// TIA Portal V17 export
// export: Created 2025-03-05T08:00:07.0490995Z, ExportSetting WithDefaults, DisplayName Totally Integrated Automation Portal, DisplayVersion V17 Update 8, DisplayName TIA Portal Openness, DisplayVersion V17 Update 8, DisplayName TIA Portal Version Control Interface, DisplayVersion V17, DisplayName SINAMICS Startdrive Advanced, DisplayVersion V17 SP2, DisplayName SINAMICS Startdrive G110M, G120, G120C, G120D, G120P, G115D, DisplayVersion V17 SP2, DisplayName SINAMICS Startdrive G130, G150, S120, S150, SINAMICS MV, S210, DisplayVersion V17 SP2, DisplayName STEP 7 Professional, DisplayVersion V17 Update 8, DisplayName SINUMERIK ONE STEP 7 Toolbox, DisplayVersion V17 Update 12, DisplayName SINUMERIK 840D sl STEP 7 Toolbox, DisplayVersion V17 Update 12, DisplayName STEP 7 Safety, DisplayVersion V17 Update 6, DisplayName WinCC Advanced, DisplayVersion V17 Update 8
FUNCTION_BLOCK "FB2002_BA_MODE"   // FB2002, LAD
{ S7_Optimized_Access := 'FALSE' }
VERSION : 0.1
// stored: AutoNumber false, IsIECCheckEnabled false, SetENOAutomatically false, UDAEnableTagReadback false
   VAR_INPUT
      OPTIONS_0 { ExternalAccessible := 'False'; ExternalVisible := 'False'; ExternalWritable := 'False'} : Byte := 2#0000_0000;   // OPTIONS BYTE 0
      BA1_BUTTON_I { ExternalAccessible := 'False'; ExternalVisible := 'False'; ExternalWritable := 'False'} : Bool;   // BA1 BUTTON INPUT
      BA2_BUTTON_I { ExternalAccessible := 'False'; ExternalVisible := 'False'; ExternalWritable := 'False'} : Bool;   // BA2 BUTTON INPUT
      BA3_BUTTON_I { ExternalAccessible := 'False'; ExternalVisible := 'False'; ExternalWritable := 'False'} : Bool;   // BA3 BUTTON INPUT
      BA5_BUTTON_I { ExternalAccessible := 'False'; ExternalVisible := 'False'; ExternalWritable := 'False'} : Bool;   // BA5 BUTTON INPUT
      SAFETY_ENABLED_W_DOOR_OPENED { ExternalAccessible := 'False'; ExternalVisible := 'False'; ExternalWritable := 'False'} : Bool;   // SAFETY ENABLED WITH DOOR OPENED (ENABLING DEVICE AND HT10 ENABLE BUTTON)
      SAFETY_GATES_CLSD_AND_LCKD { ExternalAccessible := 'False'; ExternalVisible := 'False'; ExternalWritable := 'False'} : Bool;   // SAFETY GATES CLOSED AND LOCKED
      START_SERVICES_GLOBAL { ExternalAccessible := 'False'; ExternalVisible := 'False'; ExternalWritable := 'False'} : Bool;   // START SERVICES GLOBAL
      ANY_MCH_CYCLE_RUN { ExternalAccessible := 'False'; ExternalVisible := 'False'; ExternalWritable := 'False'} : Bool;   // ANY MACHINE CYCLE RUNNING
      MCH_RESET_FAULTS { ExternalAccessible := 'False'; ExternalVisible := 'False'; ExternalWritable := 'False'} : Bool;   // MACHINE_RESET_FAULTS
   END_VAR
   VAR_OUTPUT
      NO_BA_MODE_SLCTD_WRN { ExternalAccessible := 'False'; ExternalVisible := 'False'; ExternalWritable := 'False'} : Bool;   // NO BA MODE SELECTED WARNING
      CHANGE_TO_BA1_MODE_WRN { ExternalAccessible := 'False'; ExternalVisible := 'False'; ExternalWritable := 'False'} : Bool;   // CHANGE TO BA1 MODE WARNING
      CHANGE_TO_BA2_MODE_WRN { ExternalAccessible := 'False'; ExternalVisible := 'False'; ExternalWritable := 'False'} : Bool;   // CHANGE TO BA2 MODE WARNING
      CHANGE_TO_BA3_MODE_WRN { ExternalAccessible := 'False'; ExternalVisible := 'False'; ExternalWritable := 'False'} : Bool;   // CHANGE TO BA3 MODE WARNING
      CHANGE_TO_BA5_MODE_WRN { ExternalAccessible := 'False'; ExternalVisible := 'False'; ExternalWritable := 'False'} : Bool;   // CHANGE TO BA5 MODE WARNING
      BA1_MODE_LED_O { ExternalAccessible := 'False'; ExternalVisible := 'False'; ExternalWritable := 'False'} : Bool;   // BA1 MODE BUTTON LED OUTPUT
      BA2_MODE_LED_O { ExternalAccessible := 'False'; ExternalVisible := 'False'; ExternalWritable := 'False'} : Bool;   // BA2 MODE BUTTON LED OUTPUT
      BA3_MODE_LED_O { ExternalAccessible := 'False'; ExternalVisible := 'False'; ExternalWritable := 'False'} : Bool;   // BA3 MODE BUTTON LED OUTPUT
   END_VAR
   VAR_IN_OUT
      MODE_GROUP_GENERAL_DB : "AUTO_SINGLE_SEMI_MANUAL";
      MODE_GROUP_BA_DB : "BA_MODE";
   END_VAR
   VAR_TEMP
      INPUTS_MASK : Byte;   // INPUT MASK
      O_BYTE_0 : Struct   // OPTIONS BYTE 0
         BA_BUTTONS : Bool;   // BA MODE BUTTONS OPTION
         CHANGE_MODE_SEOC_ALARM : Bool;   // CHANGE MODE SEOC ALARM OPTION
         MODE_SELECTED_MEMORY : Bool;   // MODE SELECTED MEMORY OPTION
         SPARE : Bool;
         SPARE_1 : Bool;
         SPARE_2 : Bool;
         SPARE_3 : Bool;
         SPARE_4 : Bool;
      END_STRUCT;
      DB_NUMBER : DInt;   // DB NUMBER FOR ALARM DECODING
   END_VAR
   VAR_TEMP   // added for the SCL form of the ladder/FBD networks
      _w1 : Bool;
      _w2 : Bool;
   END_VAR
BEGIN

NETWORK
TITLE = READ INSTANCE DB
      L     DINO;
      +     10#800000;
      T     #DB_NUMBER;


REGION Network 2: OPTIONS
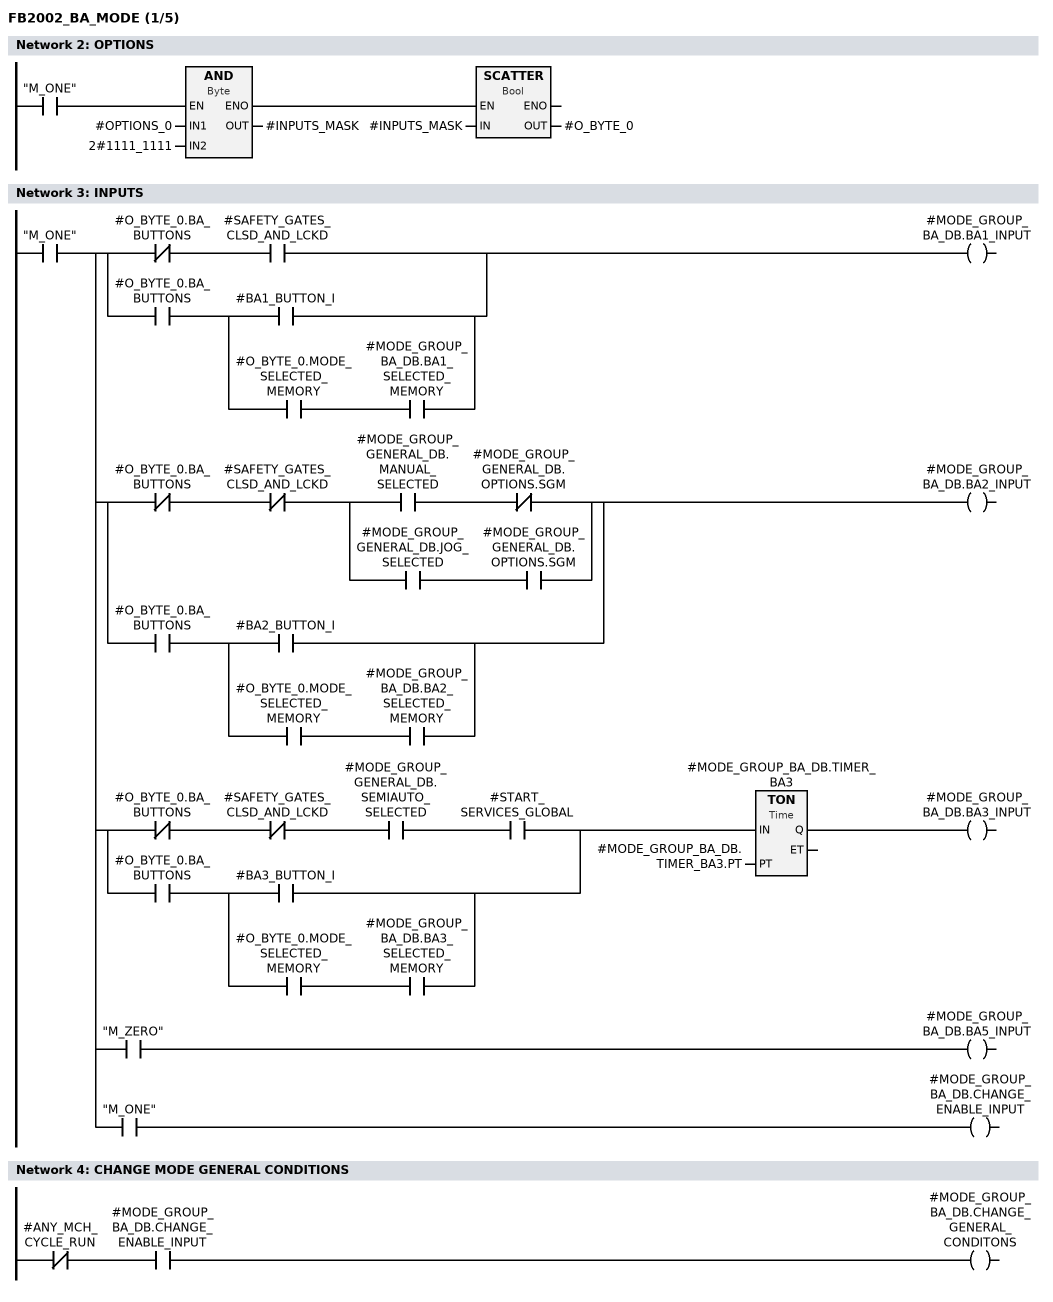
   RUNG wire#powerrail
      Contact( "M_ONE" )
      { S7_Templates := "SrcType := Byte"; S7_GenerateENO := "TRUE" } And(in1 := #OPTIONS_0, in2 := 2#1111_1111, out => #INPUTS_MASK)
      { S7_Templates := "[dest_type := Bool, src_type := Byte]" } SCATTER(IN := #INPUTS_MASK, OUT => #O_BYTE_0)
   END_RUNG
   // the same network as SCL:
   IF "M_ONE" THEN
       #INPUTS_MASK := #OPTIONS_0 AND 2#1111_1111;
       SCATTER(IN := #INPUTS_MASK, OUT => #O_BYTE_0);
   END_IF;
END_REGION

REGION Network 3: INPUTS
   RUNG wire#powerrail
      Contact( "M_ONE" )
      wire#w1
      I_Contact( #O_BYTE_0.BA_BUTTONS )
      Contact( #SAFETY_GATES_CLSD_AND_LCKD )
      wire#w2
      Coil( #MODE_GROUP_BA_DB.BA1_INPUT )
   END_RUNG
   RUNG wire#w1
      Contact( #O_BYTE_0.BA_BUTTONS )
      wire#w3
      Contact( #BA1_BUTTON_I )
   END_RUNG wire#w2
   RUNG wire#w3
      Contact( #O_BYTE_0.MODE_SELECTED_MEMORY )
      Contact( #MODE_GROUP_BA_DB.BA1_SELECTED_MEMORY )
   END_RUNG wire#w2
   RUNG wire#w1
      I_Contact( #O_BYTE_0.BA_BUTTONS )
      I_Contact( #SAFETY_GATES_CLSD_AND_LCKD )
      wire#w4
      Contact( #MODE_GROUP_GENERAL_DB.MANUAL_SELECTED )
      I_Contact( #MODE_GROUP_GENERAL_DB.OPTIONS.SGM )
      wire#w5
      Coil( #MODE_GROUP_BA_DB.BA2_INPUT )
   END_RUNG
   RUNG wire#w4
      Contact( #MODE_GROUP_GENERAL_DB.JOG_SELECTED )
      Contact( #MODE_GROUP_GENERAL_DB.OPTIONS.SGM )
   END_RUNG wire#w5
   RUNG wire#w1
      Contact( #O_BYTE_0.BA_BUTTONS )
      wire#w6
      Contact( #BA2_BUTTON_I )
   END_RUNG wire#w5
   RUNG wire#w6
      Contact( #O_BYTE_0.MODE_SELECTED_MEMORY )
      Contact( #MODE_GROUP_BA_DB.BA2_SELECTED_MEMORY )
   END_RUNG wire#w5
   RUNG wire#w1
      I_Contact( #O_BYTE_0.BA_BUTTONS )
      I_Contact( #SAFETY_GATES_CLSD_AND_LCKD )
      Contact( #MODE_GROUP_GENERAL_DB.SEMIAUTO_SELECTED )
      Contact( #START_SERVICES_GLOBAL )
      wire#w7
      { S7_Templates := "time_type := Time" } #MODE_GROUP_BA_DB.TIMER_BA3.TON(pt := #MODE_GROUP_BA_DB.TIMER_BA3.PT, et =>)
      Coil( #MODE_GROUP_BA_DB.BA3_INPUT )
   END_RUNG
   RUNG wire#w1
      Contact( #O_BYTE_0.BA_BUTTONS )
      wire#w8
      Contact( #BA3_BUTTON_I )
   END_RUNG wire#w7
   RUNG wire#w8
      Contact( #O_BYTE_0.MODE_SELECTED_MEMORY )
      Contact( #MODE_GROUP_BA_DB.BA3_SELECTED_MEMORY )
   END_RUNG wire#w7
   RUNG wire#w1
      Contact( "M_ZERO" )
      Coil( #MODE_GROUP_BA_DB.BA5_INPUT )
   END_RUNG
   RUNG wire#w1
      Contact( "M_ONE" )
      Coil( #MODE_GROUP_BA_DB.CHANGE_ENABLE_INPUT )
   END_RUNG
   // the same network as SCL:
   #MODE_GROUP_BA_DB.BA1_INPUT := "M_ONE" AND ((NOT #O_BYTE_0.BA_BUTTONS AND #SAFETY_GATES_CLSD_AND_LCKD) OR (#O_BYTE_0.BA_BUTTONS AND (#BA1_BUTTON_I OR (#O_BYTE_0.MODE_SELECTED_MEMORY AND #MODE_GROUP_BA_DB.BA1_SELECTED_MEMORY))));
   #MODE_GROUP_BA_DB.BA2_INPUT := "M_ONE" AND ((NOT #O_BYTE_0.BA_BUTTONS AND NOT #SAFETY_GATES_CLSD_AND_LCKD AND ((#MODE_GROUP_GENERAL_DB.MANUAL_SELECTED AND NOT #MODE_GROUP_GENERAL_DB.OPTIONS.SGM) OR (#MODE_GROUP_GENERAL_DB.JOG_SELECTED AND #MODE_GROUP_GENERAL_DB.OPTIONS.SGM))) OR (#O_BYTE_0.BA_BUTTONS AND (#BA2_BUTTON_I OR (#O_BYTE_0.MODE_SELECTED_MEMORY AND #MODE_GROUP_BA_DB.BA2_SELECTED_MEMORY))));
   #MODE_GROUP_BA_DB.TIMER_BA3.TON(IN := "M_ONE" AND ((NOT #O_BYTE_0.BA_BUTTONS AND NOT #SAFETY_GATES_CLSD_AND_LCKD AND #MODE_GROUP_GENERAL_DB.SEMIAUTO_SELECTED AND #START_SERVICES_GLOBAL) OR (#O_BYTE_0.BA_BUTTONS AND (#BA3_BUTTON_I OR (#O_BYTE_0.MODE_SELECTED_MEMORY AND #MODE_GROUP_BA_DB.BA3_SELECTED_MEMORY)))),
                           PT := #MODE_GROUP_BA_DB.TIMER_BA3.PT);
   #MODE_GROUP_BA_DB.BA3_INPUT := #MODE_GROUP_BA_DB.TIMER_BA3.Q;
   #MODE_GROUP_BA_DB.BA5_INPUT := "M_ONE" AND "M_ZERO";
   #MODE_GROUP_BA_DB.CHANGE_ENABLE_INPUT := "M_ONE" AND "M_ONE";
END_REGION

REGION Network 4: CHANGE MODE GENERAL CONDITIONS
   RUNG wire#powerrail
      I_Contact( #ANY_MCH_CYCLE_RUN )
      Contact( #MODE_GROUP_BA_DB.CHANGE_ENABLE_INPUT )
      Coil( #MODE_GROUP_BA_DB.CHANGE_GENERAL_CONDITONS )
   END_RUNG
   // the same network as SCL:
   #MODE_GROUP_BA_DB.CHANGE_GENERAL_CONDITONS := NOT #ANY_MCH_CYCLE_RUN AND #MODE_GROUP_BA_DB.CHANGE_ENABLE_INPUT;
END_REGION

REGION Network 5: OPERATOR HELP
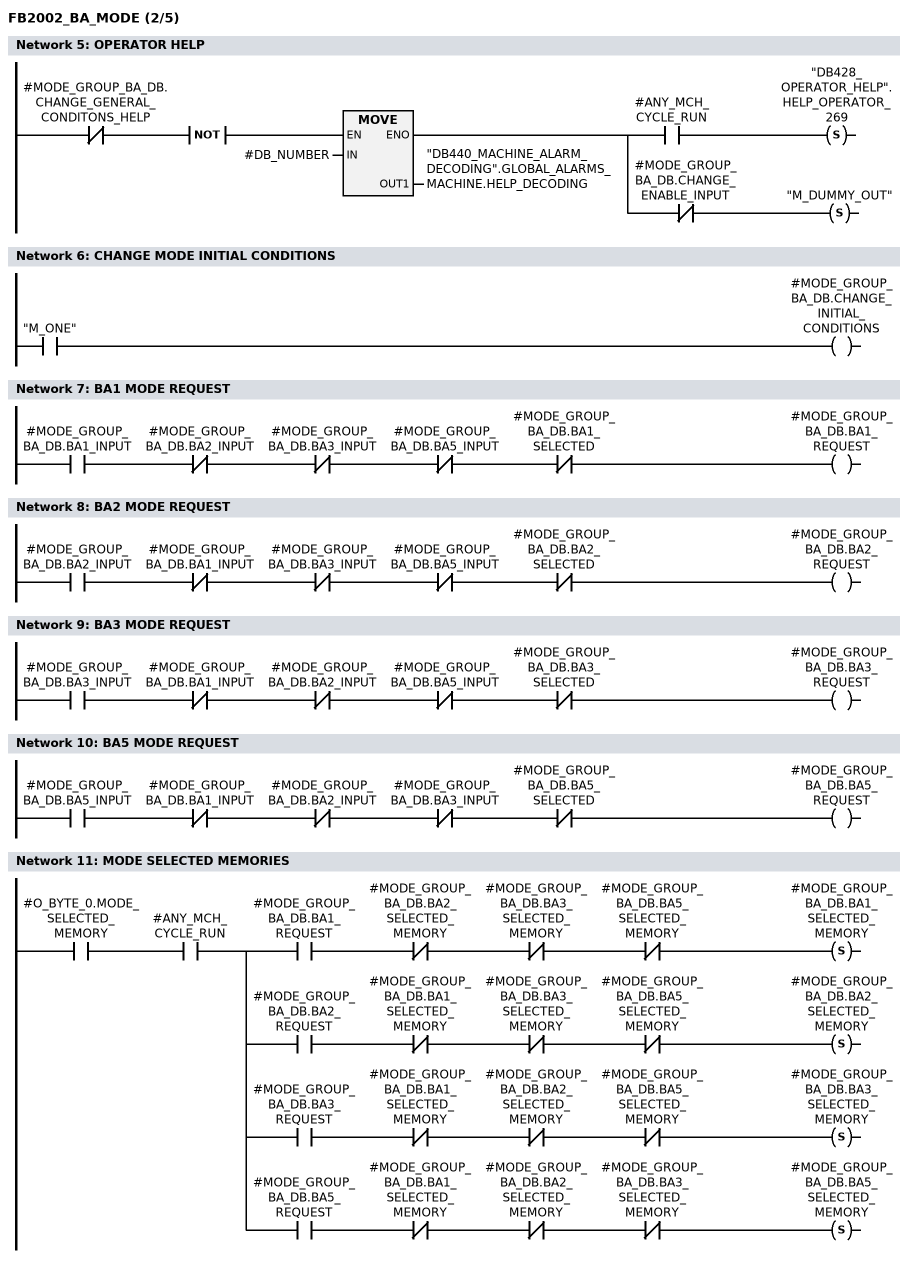
   RUNG wire#powerrail
      I_Contact( #MODE_GROUP_BA_DB.CHANGE_GENERAL_CONDITONS_HELP )
      Not()
      { S7_GenerateENO := "TRUE" } Move(in := #DB_NUMBER, out1 => "DB440_MACHINE_ALARM_DECODING".GLOBAL_ALARMS_MACHINE.HELP_DECODING)
      wire#w1
      Contact( #ANY_MCH_CYCLE_RUN )
      S_Coil( "DB428_OPERATOR_HELP".HELP_OPERATOR_269 )
   END_RUNG
   RUNG wire#w1
      I_Contact( #MODE_GROUP_BA_DB.CHANGE_ENABLE_INPUT )
      S_Coil( "M_DUMMY_OUT" )
   END_RUNG
   // the same network as SCL:
   // ENO of a box is taken as its EN; it also drops when the box reports an error
   #_w1 := NOT (NOT #MODE_GROUP_BA_DB.CHANGE_GENERAL_CONDITONS_HELP);
   IF #_w1 THEN "DB440_MACHINE_ALARM_DECODING".GLOBAL_ALARMS_MACHINE.HELP_DECODING := #DB_NUMBER; END_IF;
   IF #_w1 AND #ANY_MCH_CYCLE_RUN THEN "DB428_OPERATOR_HELP".HELP_OPERATOR_269 := TRUE; END_IF;
   IF #_w1 AND NOT #MODE_GROUP_BA_DB.CHANGE_ENABLE_INPUT THEN "M_DUMMY_OUT" := TRUE; END_IF;
END_REGION

REGION Network 6: CHANGE MODE INITIAL CONDITIONS
   RUNG wire#powerrail
      Contact( "M_ONE" )
      Coil( #MODE_GROUP_BA_DB.CHANGE_INITIAL_CONDITIONS )
   END_RUNG
   // the same network as SCL:
   #MODE_GROUP_BA_DB.CHANGE_INITIAL_CONDITIONS := "M_ONE";
END_REGION

REGION Network 7: BA1 MODE REQUEST
   RUNG wire#powerrail
      Contact( #MODE_GROUP_BA_DB.BA1_INPUT )
      I_Contact( #MODE_GROUP_BA_DB.BA2_INPUT )
      I_Contact( #MODE_GROUP_BA_DB.BA3_INPUT )
      I_Contact( #MODE_GROUP_BA_DB.BA5_INPUT )
      I_Contact( #MODE_GROUP_BA_DB.BA1_SELECTED )
      Coil( #MODE_GROUP_BA_DB.BA1_REQUEST )
   END_RUNG
   // the same network as SCL:
   #MODE_GROUP_BA_DB.BA1_REQUEST := #MODE_GROUP_BA_DB.BA1_INPUT AND NOT #MODE_GROUP_BA_DB.BA2_INPUT AND NOT #MODE_GROUP_BA_DB.BA3_INPUT AND NOT #MODE_GROUP_BA_DB.BA5_INPUT AND NOT #MODE_GROUP_BA_DB.BA1_SELECTED;
END_REGION

REGION Network 8: BA2 MODE REQUEST
   RUNG wire#powerrail
      Contact( #MODE_GROUP_BA_DB.BA2_INPUT )
      I_Contact( #MODE_GROUP_BA_DB.BA1_INPUT )
      I_Contact( #MODE_GROUP_BA_DB.BA3_INPUT )
      I_Contact( #MODE_GROUP_BA_DB.BA5_INPUT )
      I_Contact( #MODE_GROUP_BA_DB.BA2_SELECTED )
      Coil( #MODE_GROUP_BA_DB.BA2_REQUEST )
   END_RUNG
   // the same network as SCL:
   #MODE_GROUP_BA_DB.BA2_REQUEST := #MODE_GROUP_BA_DB.BA2_INPUT AND NOT #MODE_GROUP_BA_DB.BA1_INPUT AND NOT #MODE_GROUP_BA_DB.BA3_INPUT AND NOT #MODE_GROUP_BA_DB.BA5_INPUT AND NOT #MODE_GROUP_BA_DB.BA2_SELECTED;
END_REGION

REGION Network 9: BA3 MODE REQUEST
   RUNG wire#powerrail
      Contact( #MODE_GROUP_BA_DB.BA3_INPUT )
      I_Contact( #MODE_GROUP_BA_DB.BA1_INPUT )
      I_Contact( #MODE_GROUP_BA_DB.BA2_INPUT )
      I_Contact( #MODE_GROUP_BA_DB.BA5_INPUT )
      I_Contact( #MODE_GROUP_BA_DB.BA3_SELECTED )
      Coil( #MODE_GROUP_BA_DB.BA3_REQUEST )
   END_RUNG
   // the same network as SCL:
   #MODE_GROUP_BA_DB.BA3_REQUEST := #MODE_GROUP_BA_DB.BA3_INPUT AND NOT #MODE_GROUP_BA_DB.BA1_INPUT AND NOT #MODE_GROUP_BA_DB.BA2_INPUT AND NOT #MODE_GROUP_BA_DB.BA5_INPUT AND NOT #MODE_GROUP_BA_DB.BA3_SELECTED;
END_REGION

REGION Network 10: BA5 MODE REQUEST
   RUNG wire#powerrail
      Contact( #MODE_GROUP_BA_DB.BA5_INPUT )
      I_Contact( #MODE_GROUP_BA_DB.BA1_INPUT )
      I_Contact( #MODE_GROUP_BA_DB.BA2_INPUT )
      I_Contact( #MODE_GROUP_BA_DB.BA3_INPUT )
      I_Contact( #MODE_GROUP_BA_DB.BA5_SELECTED )
      Coil( #MODE_GROUP_BA_DB.BA5_REQUEST )
   END_RUNG
   // the same network as SCL:
   #MODE_GROUP_BA_DB.BA5_REQUEST := #MODE_GROUP_BA_DB.BA5_INPUT AND NOT #MODE_GROUP_BA_DB.BA1_INPUT AND NOT #MODE_GROUP_BA_DB.BA2_INPUT AND NOT #MODE_GROUP_BA_DB.BA3_INPUT AND NOT #MODE_GROUP_BA_DB.BA5_SELECTED;
END_REGION

REGION Network 11: MODE SELECTED MEMORIES
   RUNG wire#powerrail
      Contact( #O_BYTE_0.MODE_SELECTED_MEMORY )
      Contact( #ANY_MCH_CYCLE_RUN )
      wire#w1
      Contact( #MODE_GROUP_BA_DB.BA1_REQUEST )
      I_Contact( #MODE_GROUP_BA_DB.BA2_SELECTED_MEMORY )
      I_Contact( #MODE_GROUP_BA_DB.BA3_SELECTED_MEMORY )
      I_Contact( #MODE_GROUP_BA_DB.BA5_SELECTED_MEMORY )
      S_Coil( #MODE_GROUP_BA_DB.BA1_SELECTED_MEMORY )
   END_RUNG
   RUNG wire#w1
      Contact( #MODE_GROUP_BA_DB.BA2_REQUEST )
      I_Contact( #MODE_GROUP_BA_DB.BA1_SELECTED_MEMORY )
      I_Contact( #MODE_GROUP_BA_DB.BA3_SELECTED_MEMORY )
      I_Contact( #MODE_GROUP_BA_DB.BA5_SELECTED_MEMORY )
      S_Coil( #MODE_GROUP_BA_DB.BA2_SELECTED_MEMORY )
   END_RUNG
   RUNG wire#w1
      Contact( #MODE_GROUP_BA_DB.BA3_REQUEST )
      I_Contact( #MODE_GROUP_BA_DB.BA1_SELECTED_MEMORY )
      I_Contact( #MODE_GROUP_BA_DB.BA2_SELECTED_MEMORY )
      I_Contact( #MODE_GROUP_BA_DB.BA5_SELECTED_MEMORY )
      S_Coil( #MODE_GROUP_BA_DB.BA3_SELECTED_MEMORY )
   END_RUNG
   RUNG wire#w1
      Contact( #MODE_GROUP_BA_DB.BA5_REQUEST )
      I_Contact( #MODE_GROUP_BA_DB.BA1_SELECTED_MEMORY )
      I_Contact( #MODE_GROUP_BA_DB.BA2_SELECTED_MEMORY )
      I_Contact( #MODE_GROUP_BA_DB.BA3_SELECTED_MEMORY )
      S_Coil( #MODE_GROUP_BA_DB.BA5_SELECTED_MEMORY )
   END_RUNG
   // the same network as SCL:
   #_w1 := #O_BYTE_0.MODE_SELECTED_MEMORY AND #ANY_MCH_CYCLE_RUN;
   IF #_w1 AND #MODE_GROUP_BA_DB.BA1_REQUEST AND NOT #MODE_GROUP_BA_DB.BA2_SELECTED_MEMORY AND NOT #MODE_GROUP_BA_DB.BA3_SELECTED_MEMORY AND NOT #MODE_GROUP_BA_DB.BA5_SELECTED_MEMORY THEN
       #MODE_GROUP_BA_DB.BA1_SELECTED_MEMORY := TRUE;
   END_IF;
   IF #_w1 AND #MODE_GROUP_BA_DB.BA2_REQUEST AND NOT #MODE_GROUP_BA_DB.BA1_SELECTED_MEMORY AND NOT #MODE_GROUP_BA_DB.BA3_SELECTED_MEMORY AND NOT #MODE_GROUP_BA_DB.BA5_SELECTED_MEMORY THEN
       #MODE_GROUP_BA_DB.BA2_SELECTED_MEMORY := TRUE;
   END_IF;
   IF #_w1 AND #MODE_GROUP_BA_DB.BA3_REQUEST AND NOT #MODE_GROUP_BA_DB.BA1_SELECTED_MEMORY AND NOT #MODE_GROUP_BA_DB.BA2_SELECTED_MEMORY AND NOT #MODE_GROUP_BA_DB.BA5_SELECTED_MEMORY THEN
       #MODE_GROUP_BA_DB.BA3_SELECTED_MEMORY := TRUE;
   END_IF;
   IF #_w1 AND #MODE_GROUP_BA_DB.BA5_REQUEST AND NOT #MODE_GROUP_BA_DB.BA1_SELECTED_MEMORY AND NOT #MODE_GROUP_BA_DB.BA2_SELECTED_MEMORY AND NOT #MODE_GROUP_BA_DB.BA3_SELECTED_MEMORY THEN
       #MODE_GROUP_BA_DB.BA5_SELECTED_MEMORY := TRUE;
   END_IF;
END_REGION

REGION Network 12: BA1 MODE SELECTED
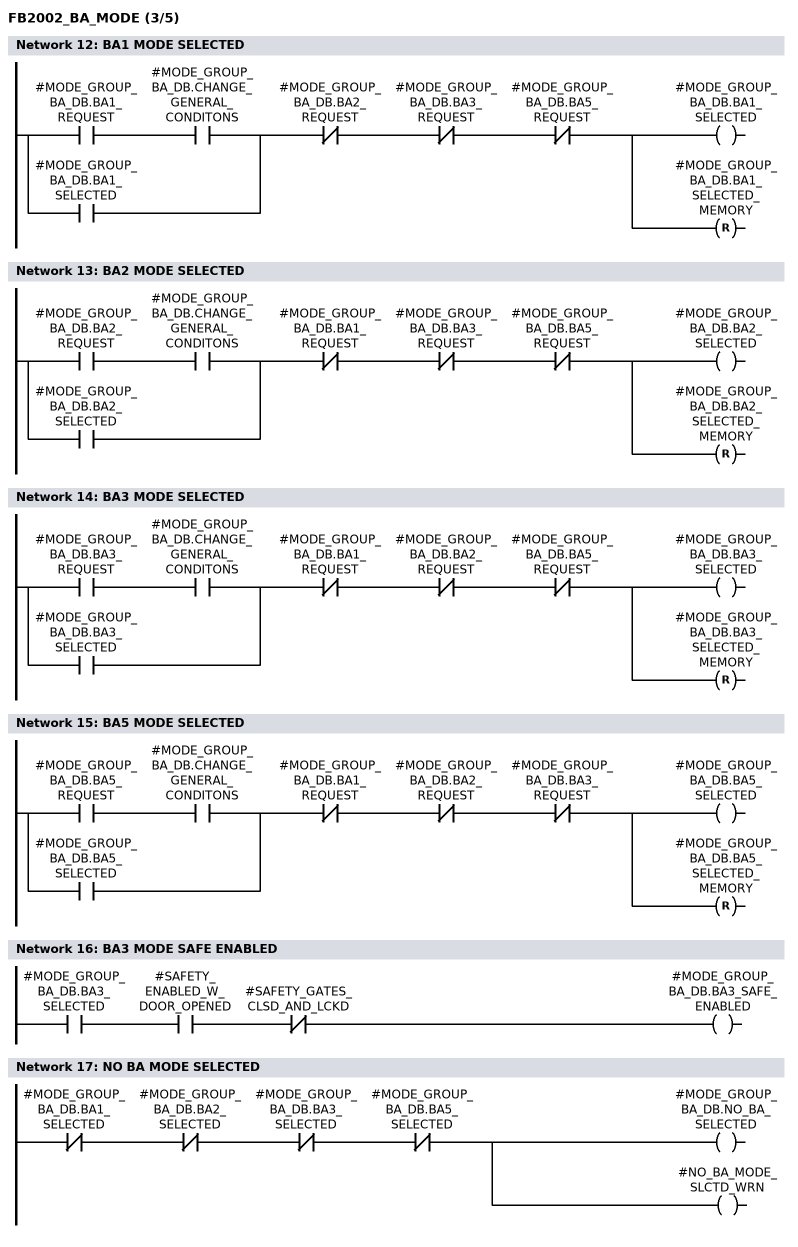
   RUNG wire#powerrail
      Contact( #MODE_GROUP_BA_DB.BA1_REQUEST )
      Contact( #MODE_GROUP_BA_DB.CHANGE_GENERAL_CONDITONS )
      wire#w1
      I_Contact( #MODE_GROUP_BA_DB.BA2_REQUEST )
      I_Contact( #MODE_GROUP_BA_DB.BA3_REQUEST )
      I_Contact( #MODE_GROUP_BA_DB.BA5_REQUEST )
      wire#w2
      Coil( #MODE_GROUP_BA_DB.BA1_SELECTED )
   END_RUNG
   RUNG wire#powerrail
      Contact( #MODE_GROUP_BA_DB.BA1_SELECTED )
   END_RUNG wire#w1
   RUNG wire#w2
      R_Coil( #MODE_GROUP_BA_DB.BA1_SELECTED_MEMORY )
   END_RUNG
   // the same network as SCL:
   #MODE_GROUP_BA_DB.BA1_SELECTED := ((#MODE_GROUP_BA_DB.BA1_REQUEST AND #MODE_GROUP_BA_DB.CHANGE_GENERAL_CONDITONS) OR #MODE_GROUP_BA_DB.BA1_SELECTED) AND NOT #MODE_GROUP_BA_DB.BA2_REQUEST AND NOT #MODE_GROUP_BA_DB.BA3_REQUEST AND NOT #MODE_GROUP_BA_DB.BA5_REQUEST;
   IF #MODE_GROUP_BA_DB.BA1_SELECTED THEN #MODE_GROUP_BA_DB.BA1_SELECTED_MEMORY := FALSE; END_IF;
END_REGION

REGION Network 13: BA2 MODE SELECTED
   RUNG wire#powerrail
      Contact( #MODE_GROUP_BA_DB.BA2_REQUEST )
      Contact( #MODE_GROUP_BA_DB.CHANGE_GENERAL_CONDITONS )
      wire#w1
      I_Contact( #MODE_GROUP_BA_DB.BA1_REQUEST )
      I_Contact( #MODE_GROUP_BA_DB.BA3_REQUEST )
      I_Contact( #MODE_GROUP_BA_DB.BA5_REQUEST )
      wire#w2
      Coil( #MODE_GROUP_BA_DB.BA2_SELECTED )
   END_RUNG
   RUNG wire#powerrail
      Contact( #MODE_GROUP_BA_DB.BA2_SELECTED )
   END_RUNG wire#w1
   RUNG wire#w2
      R_Coil( #MODE_GROUP_BA_DB.BA2_SELECTED_MEMORY )
   END_RUNG
   // the same network as SCL:
   #MODE_GROUP_BA_DB.BA2_SELECTED := ((#MODE_GROUP_BA_DB.BA2_REQUEST AND #MODE_GROUP_BA_DB.CHANGE_GENERAL_CONDITONS) OR #MODE_GROUP_BA_DB.BA2_SELECTED) AND NOT #MODE_GROUP_BA_DB.BA1_REQUEST AND NOT #MODE_GROUP_BA_DB.BA3_REQUEST AND NOT #MODE_GROUP_BA_DB.BA5_REQUEST;
   IF #MODE_GROUP_BA_DB.BA2_SELECTED THEN #MODE_GROUP_BA_DB.BA2_SELECTED_MEMORY := FALSE; END_IF;
END_REGION

REGION Network 14: BA3 MODE SELECTED
   RUNG wire#powerrail
      Contact( #MODE_GROUP_BA_DB.BA3_REQUEST )
      Contact( #MODE_GROUP_BA_DB.CHANGE_GENERAL_CONDITONS )
      wire#w1
      I_Contact( #MODE_GROUP_BA_DB.BA1_REQUEST )
      I_Contact( #MODE_GROUP_BA_DB.BA2_REQUEST )
      I_Contact( #MODE_GROUP_BA_DB.BA5_REQUEST )
      wire#w2
      Coil( #MODE_GROUP_BA_DB.BA3_SELECTED )
   END_RUNG
   RUNG wire#powerrail
      Contact( #MODE_GROUP_BA_DB.BA3_SELECTED )
   END_RUNG wire#w1
   RUNG wire#w2
      R_Coil( #MODE_GROUP_BA_DB.BA3_SELECTED_MEMORY )
   END_RUNG
   // the same network as SCL:
   #MODE_GROUP_BA_DB.BA3_SELECTED := ((#MODE_GROUP_BA_DB.BA3_REQUEST AND #MODE_GROUP_BA_DB.CHANGE_GENERAL_CONDITONS) OR #MODE_GROUP_BA_DB.BA3_SELECTED) AND NOT #MODE_GROUP_BA_DB.BA1_REQUEST AND NOT #MODE_GROUP_BA_DB.BA2_REQUEST AND NOT #MODE_GROUP_BA_DB.BA5_REQUEST;
   IF #MODE_GROUP_BA_DB.BA3_SELECTED THEN #MODE_GROUP_BA_DB.BA3_SELECTED_MEMORY := FALSE; END_IF;
END_REGION

REGION Network 15: BA5 MODE SELECTED
   RUNG wire#powerrail
      Contact( #MODE_GROUP_BA_DB.BA5_REQUEST )
      Contact( #MODE_GROUP_BA_DB.CHANGE_GENERAL_CONDITONS )
      wire#w1
      I_Contact( #MODE_GROUP_BA_DB.BA1_REQUEST )
      I_Contact( #MODE_GROUP_BA_DB.BA2_REQUEST )
      I_Contact( #MODE_GROUP_BA_DB.BA3_REQUEST )
      wire#w2
      Coil( #MODE_GROUP_BA_DB.BA5_SELECTED )
   END_RUNG
   RUNG wire#powerrail
      Contact( #MODE_GROUP_BA_DB.BA5_SELECTED )
   END_RUNG wire#w1
   RUNG wire#w2
      R_Coil( #MODE_GROUP_BA_DB.BA5_SELECTED_MEMORY )
   END_RUNG
   // the same network as SCL:
   #MODE_GROUP_BA_DB.BA5_SELECTED := ((#MODE_GROUP_BA_DB.BA5_REQUEST AND #MODE_GROUP_BA_DB.CHANGE_GENERAL_CONDITONS) OR #MODE_GROUP_BA_DB.BA5_SELECTED) AND NOT #MODE_GROUP_BA_DB.BA1_REQUEST AND NOT #MODE_GROUP_BA_DB.BA2_REQUEST AND NOT #MODE_GROUP_BA_DB.BA3_REQUEST;
   IF #MODE_GROUP_BA_DB.BA5_SELECTED THEN #MODE_GROUP_BA_DB.BA5_SELECTED_MEMORY := FALSE; END_IF;
END_REGION

REGION Network 16: BA3 MODE SAFE ENABLED
   RUNG wire#powerrail
      Contact( #MODE_GROUP_BA_DB.BA3_SELECTED )
      Contact( #SAFETY_ENABLED_W_DOOR_OPENED )
      I_Contact( #SAFETY_GATES_CLSD_AND_LCKD )
      Coil( #MODE_GROUP_BA_DB.BA3_SAFE_ENABLED )
   END_RUNG
   // the same network as SCL:
   #MODE_GROUP_BA_DB.BA3_SAFE_ENABLED := #MODE_GROUP_BA_DB.BA3_SELECTED AND #SAFETY_ENABLED_W_DOOR_OPENED AND NOT #SAFETY_GATES_CLSD_AND_LCKD;
END_REGION

REGION Network 17: NO BA MODE SELECTED
   RUNG wire#powerrail
      I_Contact( #MODE_GROUP_BA_DB.BA1_SELECTED )
      I_Contact( #MODE_GROUP_BA_DB.BA2_SELECTED )
      I_Contact( #MODE_GROUP_BA_DB.BA3_SELECTED )
      I_Contact( #MODE_GROUP_BA_DB.BA5_SELECTED )
      wire#w1
      Coil( #MODE_GROUP_BA_DB.NO_BA_SELECTED )
   END_RUNG
   RUNG wire#w1
      Coil( #NO_BA_MODE_SLCTD_WRN )
   END_RUNG
   // the same network as SCL:
   #MODE_GROUP_BA_DB.NO_BA_SELECTED := NOT #MODE_GROUP_BA_DB.BA1_SELECTED AND NOT #MODE_GROUP_BA_DB.BA2_SELECTED AND NOT #MODE_GROUP_BA_DB.BA3_SELECTED AND NOT #MODE_GROUP_BA_DB.BA5_SELECTED;
   #NO_BA_MODE_SLCTD_WRN := #MODE_GROUP_BA_DB.NO_BA_SELECTED;
END_REGION

REGION Network 18: CHANGE TO BA1 MODE ALARM
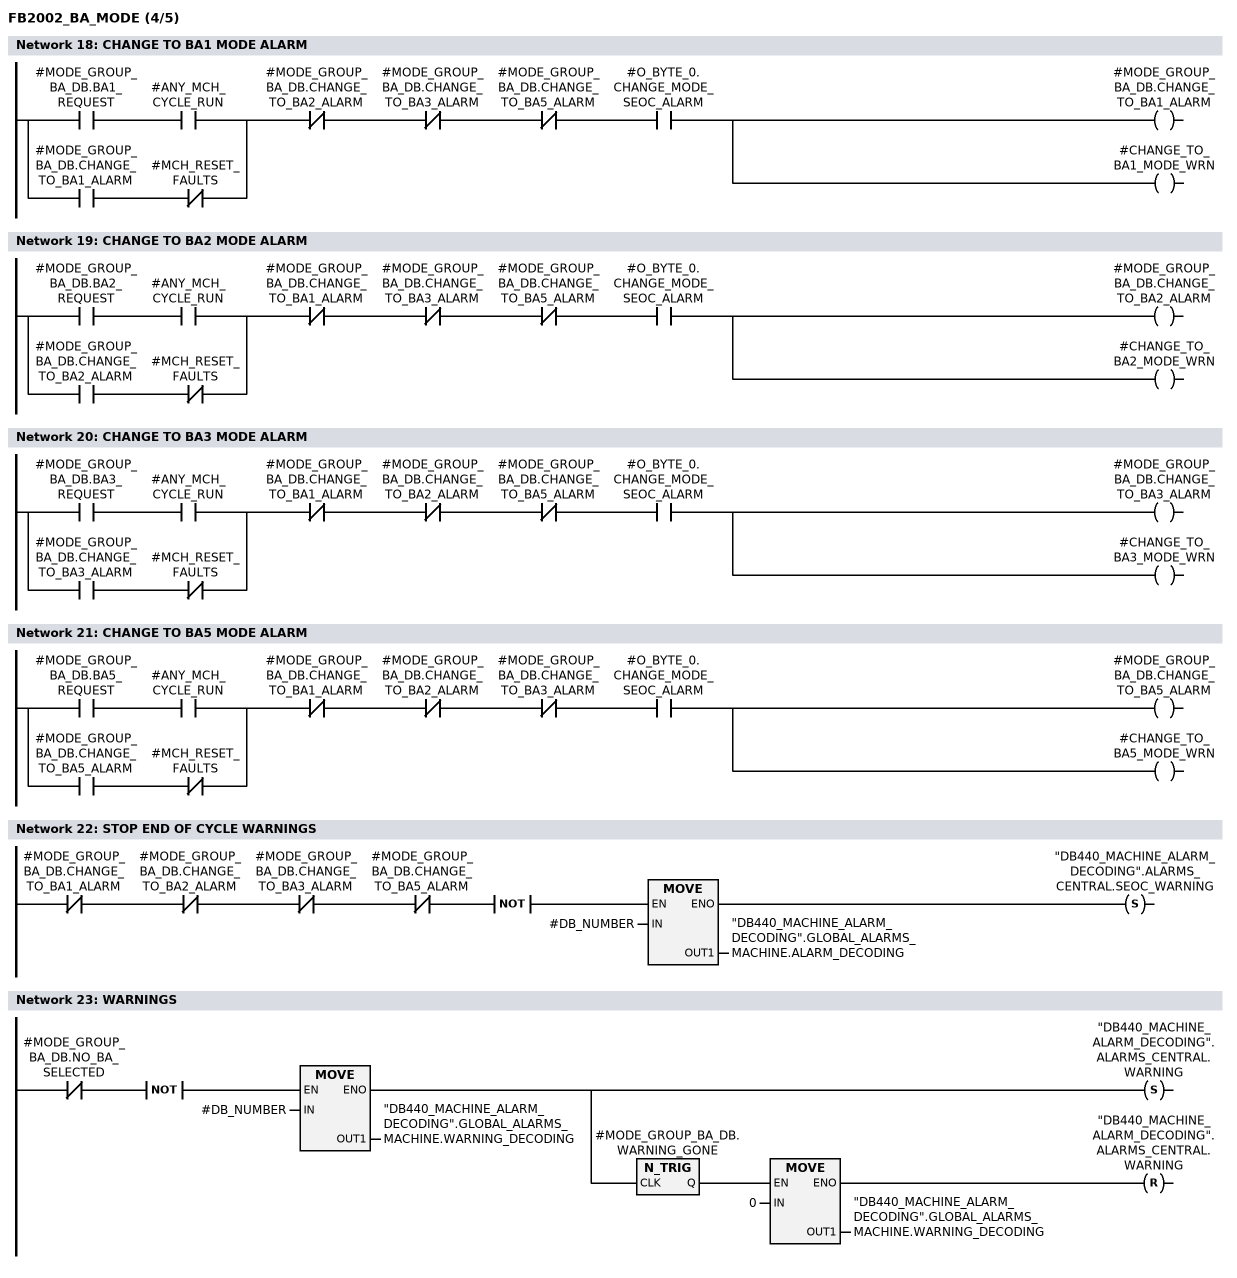
   RUNG wire#powerrail
      Contact( #MODE_GROUP_BA_DB.BA1_REQUEST )
      Contact( #ANY_MCH_CYCLE_RUN )
      wire#w1
      I_Contact( #MODE_GROUP_BA_DB.CHANGE_TO_BA2_ALARM )
      I_Contact( #MODE_GROUP_BA_DB.CHANGE_TO_BA3_ALARM )
      I_Contact( #MODE_GROUP_BA_DB.CHANGE_TO_BA5_ALARM )
      Contact( #O_BYTE_0.CHANGE_MODE_SEOC_ALARM )
      wire#w2
      Coil( #MODE_GROUP_BA_DB.CHANGE_TO_BA1_ALARM )
   END_RUNG
   RUNG wire#powerrail
      Contact( #MODE_GROUP_BA_DB.CHANGE_TO_BA1_ALARM )
      I_Contact( #MCH_RESET_FAULTS )
   END_RUNG wire#w1
   RUNG wire#w2
      Coil( #CHANGE_TO_BA1_MODE_WRN )
   END_RUNG
   // the same network as SCL:
   #MODE_GROUP_BA_DB.CHANGE_TO_BA1_ALARM := ((#MODE_GROUP_BA_DB.BA1_REQUEST AND #ANY_MCH_CYCLE_RUN) OR (#MODE_GROUP_BA_DB.CHANGE_TO_BA1_ALARM AND NOT #MCH_RESET_FAULTS)) AND NOT #MODE_GROUP_BA_DB.CHANGE_TO_BA2_ALARM AND NOT #MODE_GROUP_BA_DB.CHANGE_TO_BA3_ALARM AND NOT #MODE_GROUP_BA_DB.CHANGE_TO_BA5_ALARM AND #O_BYTE_0.CHANGE_MODE_SEOC_ALARM;
   #CHANGE_TO_BA1_MODE_WRN := #MODE_GROUP_BA_DB.CHANGE_TO_BA1_ALARM;
END_REGION

REGION Network 19: CHANGE TO BA2 MODE ALARM
   RUNG wire#powerrail
      Contact( #MODE_GROUP_BA_DB.BA2_REQUEST )
      Contact( #ANY_MCH_CYCLE_RUN )
      wire#w1
      I_Contact( #MODE_GROUP_BA_DB.CHANGE_TO_BA1_ALARM )
      I_Contact( #MODE_GROUP_BA_DB.CHANGE_TO_BA3_ALARM )
      I_Contact( #MODE_GROUP_BA_DB.CHANGE_TO_BA5_ALARM )
      Contact( #O_BYTE_0.CHANGE_MODE_SEOC_ALARM )
      wire#w2
      Coil( #MODE_GROUP_BA_DB.CHANGE_TO_BA2_ALARM )
   END_RUNG
   RUNG wire#powerrail
      Contact( #MODE_GROUP_BA_DB.CHANGE_TO_BA2_ALARM )
      I_Contact( #MCH_RESET_FAULTS )
   END_RUNG wire#w1
   RUNG wire#w2
      Coil( #CHANGE_TO_BA2_MODE_WRN )
   END_RUNG
   // the same network as SCL:
   #MODE_GROUP_BA_DB.CHANGE_TO_BA2_ALARM := ((#MODE_GROUP_BA_DB.BA2_REQUEST AND #ANY_MCH_CYCLE_RUN) OR (#MODE_GROUP_BA_DB.CHANGE_TO_BA2_ALARM AND NOT #MCH_RESET_FAULTS)) AND NOT #MODE_GROUP_BA_DB.CHANGE_TO_BA1_ALARM AND NOT #MODE_GROUP_BA_DB.CHANGE_TO_BA3_ALARM AND NOT #MODE_GROUP_BA_DB.CHANGE_TO_BA5_ALARM AND #O_BYTE_0.CHANGE_MODE_SEOC_ALARM;
   #CHANGE_TO_BA2_MODE_WRN := #MODE_GROUP_BA_DB.CHANGE_TO_BA2_ALARM;
END_REGION

REGION Network 20: CHANGE TO BA3 MODE ALARM
   RUNG wire#powerrail
      Contact( #MODE_GROUP_BA_DB.BA3_REQUEST )
      Contact( #ANY_MCH_CYCLE_RUN )
      wire#w1
      I_Contact( #MODE_GROUP_BA_DB.CHANGE_TO_BA1_ALARM )
      I_Contact( #MODE_GROUP_BA_DB.CHANGE_TO_BA2_ALARM )
      I_Contact( #MODE_GROUP_BA_DB.CHANGE_TO_BA5_ALARM )
      Contact( #O_BYTE_0.CHANGE_MODE_SEOC_ALARM )
      wire#w2
      Coil( #MODE_GROUP_BA_DB.CHANGE_TO_BA3_ALARM )
   END_RUNG
   RUNG wire#powerrail
      Contact( #MODE_GROUP_BA_DB.CHANGE_TO_BA3_ALARM )
      I_Contact( #MCH_RESET_FAULTS )
   END_RUNG wire#w1
   RUNG wire#w2
      Coil( #CHANGE_TO_BA3_MODE_WRN )
   END_RUNG
   // the same network as SCL:
   #MODE_GROUP_BA_DB.CHANGE_TO_BA3_ALARM := ((#MODE_GROUP_BA_DB.BA3_REQUEST AND #ANY_MCH_CYCLE_RUN) OR (#MODE_GROUP_BA_DB.CHANGE_TO_BA3_ALARM AND NOT #MCH_RESET_FAULTS)) AND NOT #MODE_GROUP_BA_DB.CHANGE_TO_BA1_ALARM AND NOT #MODE_GROUP_BA_DB.CHANGE_TO_BA2_ALARM AND NOT #MODE_GROUP_BA_DB.CHANGE_TO_BA5_ALARM AND #O_BYTE_0.CHANGE_MODE_SEOC_ALARM;
   #CHANGE_TO_BA3_MODE_WRN := #MODE_GROUP_BA_DB.CHANGE_TO_BA3_ALARM;
END_REGION

REGION Network 21: CHANGE TO BA5 MODE ALARM
   RUNG wire#powerrail
      Contact( #MODE_GROUP_BA_DB.BA5_REQUEST )
      Contact( #ANY_MCH_CYCLE_RUN )
      wire#w1
      I_Contact( #MODE_GROUP_BA_DB.CHANGE_TO_BA1_ALARM )
      I_Contact( #MODE_GROUP_BA_DB.CHANGE_TO_BA2_ALARM )
      I_Contact( #MODE_GROUP_BA_DB.CHANGE_TO_BA3_ALARM )
      Contact( #O_BYTE_0.CHANGE_MODE_SEOC_ALARM )
      wire#w2
      Coil( #MODE_GROUP_BA_DB.CHANGE_TO_BA5_ALARM )
   END_RUNG
   RUNG wire#powerrail
      Contact( #MODE_GROUP_BA_DB.CHANGE_TO_BA5_ALARM )
      I_Contact( #MCH_RESET_FAULTS )
   END_RUNG wire#w1
   RUNG wire#w2
      Coil( #CHANGE_TO_BA5_MODE_WRN )
   END_RUNG
   // the same network as SCL:
   #MODE_GROUP_BA_DB.CHANGE_TO_BA5_ALARM := ((#MODE_GROUP_BA_DB.BA5_REQUEST AND #ANY_MCH_CYCLE_RUN) OR (#MODE_GROUP_BA_DB.CHANGE_TO_BA5_ALARM AND NOT #MCH_RESET_FAULTS)) AND NOT #MODE_GROUP_BA_DB.CHANGE_TO_BA1_ALARM AND NOT #MODE_GROUP_BA_DB.CHANGE_TO_BA2_ALARM AND NOT #MODE_GROUP_BA_DB.CHANGE_TO_BA3_ALARM AND #O_BYTE_0.CHANGE_MODE_SEOC_ALARM;
   #CHANGE_TO_BA5_MODE_WRN := #MODE_GROUP_BA_DB.CHANGE_TO_BA5_ALARM;
END_REGION

REGION Network 22: STOP END OF CYCLE WARNINGS
   RUNG wire#powerrail
      I_Contact( #MODE_GROUP_BA_DB.CHANGE_TO_BA1_ALARM )
      I_Contact( #MODE_GROUP_BA_DB.CHANGE_TO_BA2_ALARM )
      I_Contact( #MODE_GROUP_BA_DB.CHANGE_TO_BA3_ALARM )
      I_Contact( #MODE_GROUP_BA_DB.CHANGE_TO_BA5_ALARM )
      Not()
      { S7_GenerateENO := "TRUE" } Move(in := #DB_NUMBER, out1 => "DB440_MACHINE_ALARM_DECODING".GLOBAL_ALARMS_MACHINE.ALARM_DECODING)
      S_Coil( "DB440_MACHINE_ALARM_DECODING".ALARMS_CENTRAL.SEOC_WARNING )
   END_RUNG
   // the same network as SCL:
   // ENO of a box is taken as its EN; it also drops when the box reports an error
   IF NOT (NOT #MODE_GROUP_BA_DB.CHANGE_TO_BA1_ALARM AND NOT #MODE_GROUP_BA_DB.CHANGE_TO_BA2_ALARM AND NOT #MODE_GROUP_BA_DB.CHANGE_TO_BA3_ALARM AND NOT #MODE_GROUP_BA_DB.CHANGE_TO_BA5_ALARM) THEN
       "DB440_MACHINE_ALARM_DECODING".GLOBAL_ALARMS_MACHINE.ALARM_DECODING := #DB_NUMBER;
       "DB440_MACHINE_ALARM_DECODING".ALARMS_CENTRAL.SEOC_WARNING := TRUE;
   END_IF;
END_REGION

REGION Network 23: WARNINGS
   RUNG wire#powerrail
      I_Contact( #MODE_GROUP_BA_DB.NO_BA_SELECTED )
      Not()
      Move(in := #DB_NUMBER, out1 => "DB440_MACHINE_ALARM_DECODING".GLOBAL_ALARMS_MACHINE.WARNING_DECODING)
      wire#w1
      S_Coil( "DB440_MACHINE_ALARM_DECODING".ALARMS_CENTRAL.WARNING )
   END_RUNG
   RUNG wire#w1
      N_Trig( #MODE_GROUP_BA_DB.WARNING_GONE )
      Move(in := 0, out1 => "DB440_MACHINE_ALARM_DECODING".GLOBAL_ALARMS_MACHINE.WARNING_DECODING)
      R_Coil( "DB440_MACHINE_ALARM_DECODING".ALARMS_CENTRAL.WARNING )
   END_RUNG
   // the same network as SCL:
   #_w1 := NOT (NOT #MODE_GROUP_BA_DB.NO_BA_SELECTED);
   IF #_w1 THEN
       "DB440_MACHINE_ALARM_DECODING".GLOBAL_ALARMS_MACHINE.WARNING_DECODING := #DB_NUMBER;
       "DB440_MACHINE_ALARM_DECODING".ALARMS_CENTRAL.WARNING := TRUE;
   END_IF;
   #_w2 := NOT #_w1 AND #MODE_GROUP_BA_DB.WARNING_GONE;   // falling edge
   #MODE_GROUP_BA_DB.WARNING_GONE := #_w1;
   IF #_w2 THEN
       "DB440_MACHINE_ALARM_DECODING".GLOBAL_ALARMS_MACHINE.WARNING_DECODING := 0;
       "DB440_MACHINE_ALARM_DECODING".ALARMS_CENTRAL.WARNING := FALSE;
   END_IF;
END_REGION

REGION Network 24: CHANGE MODE GENERAL CONDITIONS HELP
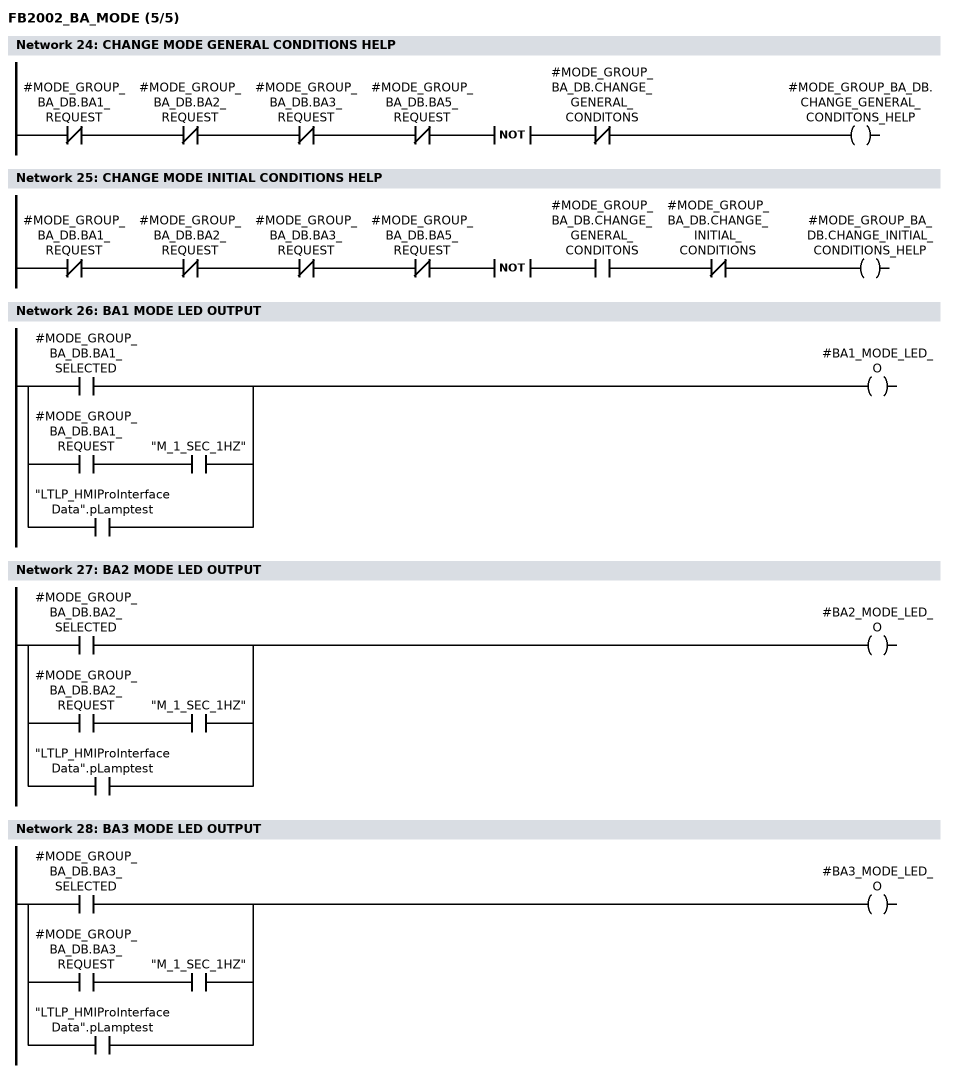
   RUNG wire#powerrail
      I_Contact( #MODE_GROUP_BA_DB.BA1_REQUEST )
      I_Contact( #MODE_GROUP_BA_DB.BA2_REQUEST )
      I_Contact( #MODE_GROUP_BA_DB.BA3_REQUEST )
      I_Contact( #MODE_GROUP_BA_DB.BA5_REQUEST )
      Not()
      I_Contact( #MODE_GROUP_BA_DB.CHANGE_GENERAL_CONDITONS )
      Coil( #MODE_GROUP_BA_DB.CHANGE_GENERAL_CONDITONS_HELP )
   END_RUNG
   // the same network as SCL:
   #MODE_GROUP_BA_DB.CHANGE_GENERAL_CONDITONS_HELP := NOT (NOT #MODE_GROUP_BA_DB.BA1_REQUEST AND NOT #MODE_GROUP_BA_DB.BA2_REQUEST AND NOT #MODE_GROUP_BA_DB.BA3_REQUEST AND NOT #MODE_GROUP_BA_DB.BA5_REQUEST) AND NOT #MODE_GROUP_BA_DB.CHANGE_GENERAL_CONDITONS;
END_REGION

REGION Network 25: CHANGE MODE INITIAL CONDITIONS HELP
   RUNG wire#powerrail
      I_Contact( #MODE_GROUP_BA_DB.BA1_REQUEST )
      I_Contact( #MODE_GROUP_BA_DB.BA2_REQUEST )
      I_Contact( #MODE_GROUP_BA_DB.BA3_REQUEST )
      I_Contact( #MODE_GROUP_BA_DB.BA5_REQUEST )
      Not()
      Contact( #MODE_GROUP_BA_DB.CHANGE_GENERAL_CONDITONS )
      I_Contact( #MODE_GROUP_BA_DB.CHANGE_INITIAL_CONDITIONS )
      Coil( #MODE_GROUP_BA_DB.CHANGE_INITIAL_CONDITIONS_HELP )
   END_RUNG
   // the same network as SCL:
   #MODE_GROUP_BA_DB.CHANGE_INITIAL_CONDITIONS_HELP := NOT (NOT #MODE_GROUP_BA_DB.BA1_REQUEST AND NOT #MODE_GROUP_BA_DB.BA2_REQUEST AND NOT #MODE_GROUP_BA_DB.BA3_REQUEST AND NOT #MODE_GROUP_BA_DB.BA5_REQUEST) AND #MODE_GROUP_BA_DB.CHANGE_GENERAL_CONDITONS AND NOT #MODE_GROUP_BA_DB.CHANGE_INITIAL_CONDITIONS;
END_REGION

REGION Network 26: BA1 MODE LED OUTPUT
   RUNG wire#powerrail
      Contact( #MODE_GROUP_BA_DB.BA1_SELECTED )
      wire#w1
      Coil( #BA1_MODE_LED_O )
   END_RUNG
   RUNG wire#powerrail
      Contact( #MODE_GROUP_BA_DB.BA1_REQUEST )
      Contact( "M_1_SEC_1HZ" )
   END_RUNG wire#w1
   RUNG wire#powerrail
      Contact( "LTLP_HMIProInterfaceData".pLamptest )
   END_RUNG wire#w1
   // the same network as SCL:
   #BA1_MODE_LED_O := #MODE_GROUP_BA_DB.BA1_SELECTED OR (#MODE_GROUP_BA_DB.BA1_REQUEST AND "M_1_SEC_1HZ") OR "LTLP_HMIProInterfaceData".pLamptest;
END_REGION

REGION Network 27: BA2 MODE LED OUTPUT
   RUNG wire#powerrail
      Contact( #MODE_GROUP_BA_DB.BA2_SELECTED )
      wire#w1
      Coil( #BA2_MODE_LED_O )
   END_RUNG
   RUNG wire#powerrail
      Contact( #MODE_GROUP_BA_DB.BA2_REQUEST )
      Contact( "M_1_SEC_1HZ" )
   END_RUNG wire#w1
   RUNG wire#powerrail
      Contact( "LTLP_HMIProInterfaceData".pLamptest )
   END_RUNG wire#w1
   // the same network as SCL:
   #BA2_MODE_LED_O := #MODE_GROUP_BA_DB.BA2_SELECTED OR (#MODE_GROUP_BA_DB.BA2_REQUEST AND "M_1_SEC_1HZ") OR "LTLP_HMIProInterfaceData".pLamptest;
END_REGION

REGION Network 28: BA3 MODE LED OUTPUT
   RUNG wire#powerrail
      Contact( #MODE_GROUP_BA_DB.BA3_SELECTED )
      wire#w1
      Coil( #BA3_MODE_LED_O )
   END_RUNG
   RUNG wire#powerrail
      Contact( #MODE_GROUP_BA_DB.BA3_REQUEST )
      Contact( "M_1_SEC_1HZ" )
   END_RUNG wire#w1
   RUNG wire#powerrail
      Contact( "LTLP_HMIProInterfaceData".pLamptest )
   END_RUNG wire#w1
   // the same network as SCL:
   #BA3_MODE_LED_O := #MODE_GROUP_BA_DB.BA3_SELECTED OR (#MODE_GROUP_BA_DB.BA3_REQUEST AND "M_1_SEC_1HZ") OR "LTLP_HMIProInterfaceData".pLamptest;
END_REGION
END_FUNCTION_BLOCK
